// TIA Portal V20 export
DATA_BLOCK "2300_EmptyCamData"   // DB121
// stored: MemoryReserve 100
   VAR
      EmptyPoint : Array[1..10000] of TO_Cam_Struct_PointData;
      EmptySegment { S7_SetPoint := 'True'} : Array[1..50] of TO_Cam_Struct_SegmentData;
   END_VAR
BEGIN
END_DATA_BLOCK
